FUNCTION_BLOCK FB_HMI_DELAY_LINES EXTENDS FB_HMI_COMPONENT
VAR_INPUT
END_VAR
VAR_OUTPUT
END_VAR
VAR
END_VAR
VAR_IN_OUT
	{attribute 'OPC.UA.DA' := '0'}
	fbInstance		: FB_NOTT_DELAY_LINES;


END_VAR


fbHealthStatus( 
				bIsEnabled:= TRUE, 
				bIsGood := NOT fbInstance.stat.bError,
				bHasWarning := fbInstance.stat.bWarning
				);
				
fbBusyStatus(
				bIsBusy := fbInstance.stat.bBusy,
				bIsEnabled := TRUE);
				
M_UpdateStatusColor();

END_FUNCTION_BLOCK

(* stored: Version 1.1.0.1, ProductVersion 3.1.4024.14
   POU FB_HMI_DELAY_LINES: Id {aea38926-fd35-46d0-8f1b-8897bc7dd10c}, SpecialFunc None *)
